{attribute 'Tc2GvlVarNames'}
VAR_GLOBAL
	DevState_Ethercat		AT %I*:UINT:=0;
	
	Tab_Affichage							:ARRAY[0..29]OF INT;
	n										:INT:=0;
	Tableau_Etat_Ethercat					:ARRAY[0..200] OF ST_EcSlaveState;
	Tableau_Esclaves						:ARRAY[0..200] OF ST_EcSlaveConfigData;	(*Tableau dans lequel le pointeur de la fb viendra écrire les informations de tous les éléments éthercat du réseaux *)

END_VAR

(* stored: Version 1.1.0.1, ProductVersion 3.1.4024.15
   GVL IO_Glob_Status_ethercat: Id {7dc58870-c29f-4443-a3b3-5e7150d534ae} *)
